Staubli VAL3: nullKey.pgx

public program nullKey(num& x_nKey[])
begin
  wait(getKey()==-1)
  x_nKey=0
end
